// TIA Portal V19 export
FUNCTION_BLOCK "AreaGen_SafetyInterface_FB"   // FB6, LAD
// stored: Access Published, MemoryReserve 100, SetENOAutomatically false
   VAR_INPUT
      AreaInterface1 : "AreaInterface";
      AreaInterface2 : "AreaInterface";
      AreaInterface3 : "AreaInterface";
      AreaInterface4 : "AreaInterface";
   END_VAR
   VAR_OUTPUT
      MachineInterface1 : "MachineInterface";
      MachineInterface2 : "MachineInterface";
      MachineInterface3 : "MachineInterface";
      MachineInterface4 : "MachineInterface";
   END_VAR
   VAR
      Alarm : Struct
         G { ExternalAccessible := 'False'; ExternalVisible := 'False'; ExternalWritable := 'False'} : Struct
            EStop : Struct
               Area01 : Bool;
               Area02 : Bool;
               Area03 : Bool;
            END_STRUCT;
            FIO_Passivation : Struct
               Module_412A1 : Bool;
               Module_468A1 : Bool;
               Module_468A2 : Bool;
               Module_468A3 : Bool;
               Module_468A4 : Bool;
               Module_468A5 : Bool;
               Module_468A6 : Bool;
               Module_468A7 : Bool;
               Module_468A8 : Bool;
               Module_470A1 : Bool;
               Module_470A2 : Bool;
               Module_471A1 : Bool;
               Module_471A2 : Bool;
               Module_472A1 : Bool;
               Module_495A1 : Bool;
               Module_495A2 : Bool;
               Module_495A3 : Bool;
               Module_515A1 : Bool;
               Module_515A2 : Bool;
               Module_535A1 : Bool;
               Module_535A2 : Bool;
               Module_536A1 : Bool;
               Module_555A1 : Bool;
               Module_556A1 : Bool;
            END_STRUCT;
            FDBACK_Error : Struct
               F_Valve_Air_Gen_Contattore : Bool;
               F_Valve_Air_Gen_Cursore : Bool;
            END_STRUCT;
         END_STRUCT;
         Area01 { ExternalAccessible := 'False'; ExternalVisible := 'False'; ExternalWritable := 'False'} : Struct
            FDBACK_Error : Struct
               SafetyValve_CoilCar : Struct
                  FDO_FBK_ERROR : Bool;
                  EV_SAFETY_FBK_WARNING : Bool;
               END_STRUCT;
               SafetyValve_DecoilersHorizRotation : Struct
                  FDO_FBK_ERROR : Bool;
                  EV_SAFETY_FBK_WARNING : Bool;
               END_STRUCT;
               SafetyValve_Decoiler1 : Struct
                  FDO_FBK_ERROR : Bool;
                  EV_SAFETY_FBK_WARNING : Bool;
               END_STRUCT;
               SafetyValve_Decoiler2 : Struct
                  FDO_FBK_ERROR : Bool;
                  EV_SAFETY_FBK_WARNING : Bool;
               END_STRUCT;
               SafetyValve_Peeler : Struct
                  FDO_FBK_ERROR : Bool;
                  EV_SAFETY_FBK_WARNING : Bool;
               END_STRUCT;
               SafetyValve_JB_Cut_Rest : Struct
                  FDO_FBK_ERROR : Bool;
                  EV_SAFETY_FBK_WARNING : Bool;
               END_STRUCT;
               SafetyValve_JB_Cut_Work : Struct
                  FDO_FBK_ERROR : Bool;
                  EV_SAFETY_FBK_WARNING : Bool;
               END_STRUCT;
               HU_Decoilers_Motor_F_Contactor : Bool;
               HU_Area01_Motor_F_Contactor : Bool;
            END_STRUCT;
            S120_SafetyFaultActive : Struct
               CoilCar : Bool;
               DecoilersTranslation : Bool;
               Decoiler1 : Bool;
               Decoiler2 : Bool;
               Straightener : Bool;
               JBTorch : Bool;
               JBPinchRoll : Bool;
            END_STRUCT;
            UnathorizedOpen : Struct
               D01 : Bool;
               D02 : Bool;
               D03 : Bool;
               D04 : Bool;
               D05 : Bool;
               D07 : Bool;
            END_STRUCT;
         END_STRUCT;
         Area02 { ExternalAccessible := 'False'; ExternalVisible := 'False'; ExternalWritable := 'False'} : Struct
            FDBACK_Error : Struct
               F_Contactor_Rollformer_CambioFormato : Bool;
               F_Contactor_FinalCut_HU_Motor : Bool;
               F_Contactor_FinalCut_HU_Valve : Bool;
            END_STRUCT;
            S120_SafetyFaultActive : Struct
               Cassetta1_OP : Bool;
               Cassetta1_MOT : Bool;
               Cassetta2_OP : Bool;
               Cassetta2_MOT : Bool;
               Cassetta3_OP : Bool;
               Cassetta3_MOT : Bool;
               Rollformer : Bool;
               FAK_PusherAx : Bool;
               FlyCarriage : Bool;
               AccRolls1 : Bool;
               AccRolls2 : Bool;
               AccRolls3 : Bool;
            END_STRUCT;
            UnathorizedOpen : Struct
               D10 : Bool;
               D11 : Bool;
               D12 : Bool;
               D14 : Bool;
               D15 : Bool;
               D16 : Bool;
               D18 : Bool;
            END_STRUCT;
            PathTest_Rollformer : Bool;
         END_STRUCT;
         Area03_04 { ExternalAccessible := 'False'; ExternalVisible := 'False'; ExternalWritable := 'False'} : Struct
            FDBACK_Error : Struct
               F_Valve_Air_A0301_A0302_Contattore : Bool;
               F_Valve_Air_A0301_A0302_Cursore : Bool;
               F_Contactor_CambioFormato_Bordatrice : Bool;
               F_Contactor_Valvole_Pareggiatore_Testa : Bool;
               F_Contactor_Valvole_Pareggiatore_Coda : Bool;
               F_Valve_Air_A0302_A0303_Contattore : Bool;
               F_Valve_Air_A0302_A0303_Cursore : Bool;
               F_Valve_Air_A0304_Contattore : Bool;
               F_Valve_Air_A0304_Cursore : Bool;
            END_STRUCT;
            S120_SafetyFaultActive : Struct
               Trasporto : Bool;
               Ribaltatore : Bool;
               Spintore : Bool;
               Bordatrice : Bool;
               Rulliera_1 : Bool;
               Rulliera_2 : Bool;
               PareggiatoreCoda : Bool;
               PareggiatoreTesta : Bool;
               ManipolatoreCoda : Bool;
               ManipolatoreTesta : Bool;
               SpallaCoda : Bool;
               SpallaTesta : Bool;
               TraslazioneCoda : Bool;
               TraslazioneTesta : Bool;
               SollevamentoCoda : Bool;
               SollevamentoTesta : Bool;
               SostegnoAntiribCoda : Bool;
               SostegnoAntiribTesta : Bool;
               NavettaTesta : Bool;
               NavettaCoda : Bool;
            END_STRUCT;
            UnathorizedOpen : Struct
               D19 : Bool;
               D20 : Bool;
               D21 : Bool;
               D22 : Bool;
               D24 : Bool;
               D25 : Bool;
               D27 : Bool;
            END_STRUCT;
            PathTest_Bordatrice : Bool;
         END_STRUCT;
      END_STRUCT;
      Warning : Struct
         G { ExternalAccessible := 'False'; ExternalVisible := 'False'; ExternalWritable := 'False'} : Struct
            EStop_CC : Bool;
            EStop_A01_Front : Bool;
            EStop_A01_Rear : Bool;
            EStop_A02_Front : Bool;
            EStop_A02_Rear : Bool;
            EStop_A03_Front_1 : Bool;
            EStop_A03_Front_2 : Bool;
            EStop_A03_Front_3 : Bool;
            EStop_A03_Rear_1 : Bool;
            EStop_A03_Rear_2 : Bool;
            EStop_A03_Rear_3 : Bool;
         END_STRUCT;
         Area01 { ExternalAccessible := 'False'; ExternalVisible := 'False'; ExternalWritable := 'False'} : Struct
            Selectors : Struct
               Maintenance_MB1 : Bool;
            END_STRUCT;
            DoorOpened : Struct
               D01 : Bool;
               D02 : Bool;
               D03 : Bool;
               D04 : Bool;
               D05 : Bool;
               D06 : Bool;   // NOt EXIST
               D07 : Bool;
            END_STRUCT;
            DoorOpenRequest : Struct
               D01 : Bool;
               D02 : Bool;
               D03 : Bool;
               D04 : Bool;
               D05 : Bool;
               D06 : Bool;   // NOt EXIST
               D07 : Bool;
            END_STRUCT;
            DoorNotLocked : Struct
               D04 : Bool;
               D05 : Bool;
               D07 : Bool;
            END_STRUCT;
         END_STRUCT;
         Area02 { ExternalAccessible := 'False'; ExternalVisible := 'False'; ExternalWritable := 'False'} : Struct
            Selectors : Struct
               Maintenance_MB2 : Bool;
            END_STRUCT;
            Feedback : Struct
               F_Valve_Area02_HU : Bool;
            END_STRUCT;
            DoorOpened : Struct
               D10 : Bool;
               D11 : Bool;
               D12 : Bool;
               D14 : Bool;
               D15 : Bool;
               D16 : Bool;
               D18 : Bool;
            END_STRUCT;
            DoorOpenRequest : Struct
               D10 : Bool;
               D11 : Bool;
               D12 : Bool;
               D14 : Bool;
               D15 : Bool;
               D16 : Bool;
               D18 : Bool;
            END_STRUCT;
            PathTest_Rollformer : Bool;
         END_STRUCT;
         Area03_04 { ExternalAccessible := 'False'; ExternalVisible := 'False'; ExternalWritable := 'False'} : Struct
            Selectors : Struct
               Maintenance_MB3 : Bool;
            END_STRUCT;
            DoorOpened : Struct
               D18 : Bool;
               D19 : Bool;
               D20 : Bool;
               D21 : Bool;
               D22 : Bool;
               D24 : Bool;
               D25 : Bool;
               D27 : Bool;
            END_STRUCT;
            DoorOpenRequest : Struct
               D16 : Bool;
               D18 : Bool;
               D19 : Bool;
               D20 : Bool;
               D21 : Bool;
               D22 : Bool;
               D24 : Bool;
               D25 : Bool;
               D27 : Bool;
            END_STRUCT;
            DoorNotLocked : Struct
               D16 : Bool;
               D19 : Bool;
               D20 : Bool;
               D21 : Bool;
               D25 : Bool;
               D27 : Bool;
            END_STRUCT;
            PathTest_Bodatrice : Bool;
         END_STRUCT;
         NoAutReady : Bool;
      END_STRUCT;
      HMI : Struct
         PbResetEletricDoor : Bool;
         LpResetEletricDoor : Bool;
      END_STRUCT;
      TON_ResetEletricDoor : TON_TIME;
      AreaG_Safety { S7_SetPoint := 'True'} : "AreaG_SafetyInterface_FB";
      Area01_Safety { S7_SetPoint := 'True'} : "Area01_SafetyInterface_FB";
      Area02_Safety { S7_SetPoint := 'True'} : "Area02_SafetyInterface_FB";
      Area03_04_Safety { S7_SetPoint := 'True'} : "Area03_04_SafetyInterface_FB";
   END_VAR
   VAR_TEMP
      Rst : Bool;
      WarningPresebce : Bool;
   END_VAR
BEGIN

REGION Network 1: Reset alarms
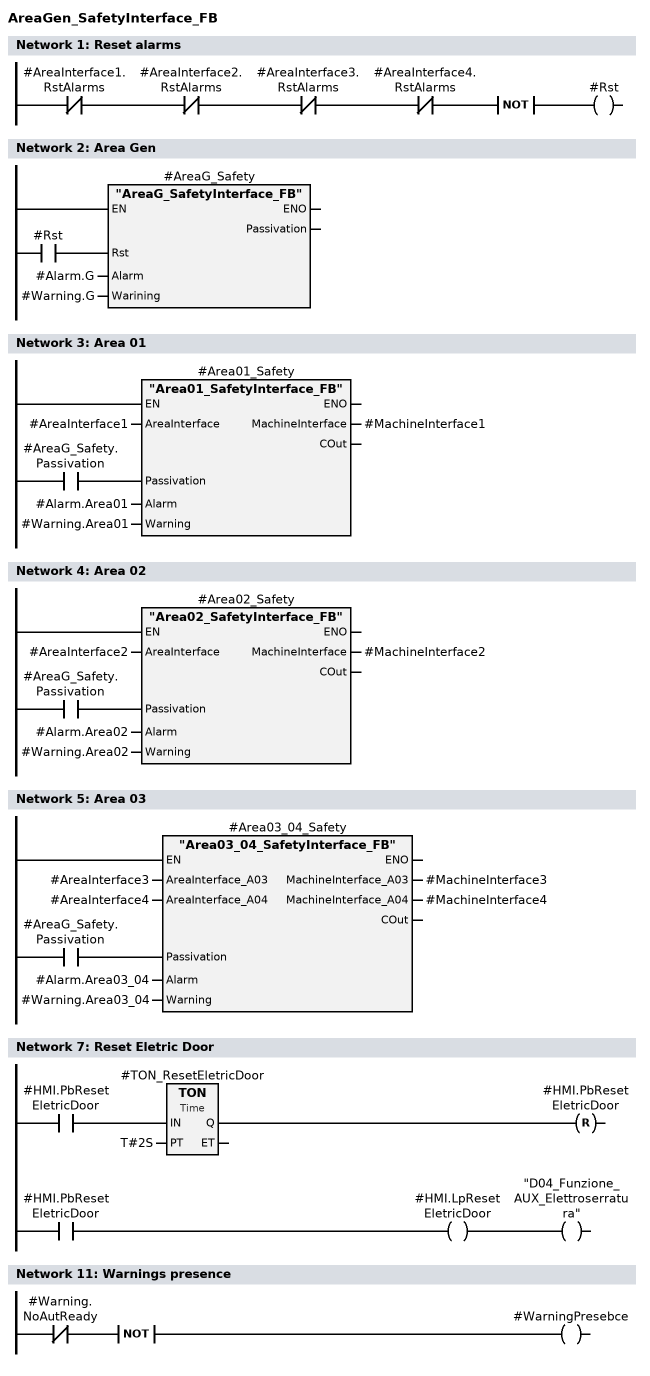
   RUNG wire#powerrail
      I_Contact( #AreaInterface1.RstAlarms )
      I_Contact( #AreaInterface2.RstAlarms )
      I_Contact( #AreaInterface3.RstAlarms )
      I_Contact( #AreaInterface4.RstAlarms )
      Not()
      Coil( #Rst )
   END_RUNG
   // the same network as SCL:
   #Rst := NOT (NOT #AreaInterface1.RstAlarms AND NOT #AreaInterface2.RstAlarms AND NOT #AreaInterface3.RstAlarms AND NOT #AreaInterface4.RstAlarms);
END_REGION

REGION Network 2: Area Gen
   RUNG wire#powerrail
      #AreaG_Safety(Rst := wire#w1, Alarm := #Alarm.G, Warining := #Warning.G, Passivation =>)
   END_RUNG
   RUNG wire#powerrail
      Contact( #Rst )
   END_RUNG wire#w1
   // the same network as SCL:
   #AreaG_Safety(Rst := #Rst, Alarm := #Alarm.G, Warining := #Warning.G);   // "AreaG_SafetyInterface_FB"
END_REGION

REGION Network 3: Area 01
   RUNG wire#powerrail
      #Area01_Safety(Passivation := wire#w1, AreaInterface := #AreaInterface1, Alarm := #Alarm.Area01, Warning := #Warning.Area01, MachineInterface => #MachineInterface1, COut =>)
   END_RUNG
   RUNG wire#powerrail
      Contact( #AreaG_Safety.Passivation )
   END_RUNG wire#w1
   // the same network as SCL:
   #Area01_Safety(AreaInterface := #AreaInterface1,   // "Area01_SafetyInterface_FB"
                  Passivation := #AreaG_Safety.Passivation,
                  Alarm := #Alarm.Area01,
                  Warning := #Warning.Area01,
                  MachineInterface => #MachineInterface1);
END_REGION

REGION Network 4: Area 02
   RUNG wire#powerrail
      #Area02_Safety(Passivation := wire#w1, AreaInterface := #AreaInterface2, Alarm := #Alarm.Area02, Warning := #Warning.Area02, MachineInterface => #MachineInterface2, COut =>)
   END_RUNG
   RUNG wire#powerrail
      Contact( #AreaG_Safety.Passivation )
   END_RUNG wire#w1
   // the same network as SCL:
   #Area02_Safety(AreaInterface := #AreaInterface2,   // "Area02_SafetyInterface_FB"
                  Passivation := #AreaG_Safety.Passivation,
                  Alarm := #Alarm.Area02,
                  Warning := #Warning.Area02,
                  MachineInterface => #MachineInterface2);
END_REGION

REGION Network 5: Area 03
   RUNG wire#powerrail
      #Area03_04_Safety(Passivation := wire#w1, AreaInterface_A03 := #AreaInterface3, AreaInterface_A04 := #AreaInterface4, Alarm := #Alarm.Area03_04, Warning := #Warning.Area03_04, MachineInterface_A03 => #MachineInterface3, MachineInterface_A04 => #MachineInterface4, COut =>)
   END_RUNG
   RUNG wire#powerrail
      Contact( #AreaG_Safety.Passivation )
   END_RUNG wire#w1
   // the same network as SCL:
   #Area03_04_Safety(AreaInterface_A03 := #AreaInterface3,   // "Area03_04_SafetyInterface_FB"
                     AreaInterface_A04 := #AreaInterface4,
                     Passivation := #AreaG_Safety.Passivation,
                     Alarm := #Alarm.Area03_04,
                     Warning := #Warning.Area03_04,
                     MachineInterface_A03 => #MachineInterface3,
                     MachineInterface_A04 => #MachineInterface4);
END_REGION

REGION Network 7: Reset Eletric Door
   RUNG wire#powerrail
      Contact( #HMI.PbResetEletricDoor )
      { S7_Templates := "time_type := Time" } #TON_ResetEletricDoor.TON(pt := T#2S, et =>)
      R_Coil( #HMI.PbResetEletricDoor )
   END_RUNG
   RUNG wire#powerrail
      Contact( #HMI.PbResetEletricDoor )
      Coil( #HMI.LpResetEletricDoor )
      Coil( "D04_Funzione_AUX_Elettroserratura" )
   END_RUNG
   // the same network as SCL:
   #TON_ResetEletricDoor(IN := #HMI.PbResetEletricDoor, PT := T#2S);   // TON
   IF #TON_ResetEletricDoor.Q THEN #HMI.PbResetEletricDoor := FALSE; END_IF;
   #HMI.LpResetEletricDoor := #HMI.PbResetEletricDoor;
   "D04_Funzione_AUX_Elettroserratura" := #HMI.PbResetEletricDoor;
END_REGION

REGION Network 9: <<< MACHINE STATUS >>>
END_REGION

REGION Network 10: Standstill
END_REGION

REGION Network 11: Warnings presence
   RUNG wire#powerrail
      I_Contact( #Warning.NoAutReady )
      Not()
      Coil( #WarningPresebce )
   END_RUNG
   // the same network as SCL:
   #WarningPresebce := NOT (NOT #Warning.NoAutReady);
END_REGION

REGION Network 12 (SCL): Collect machine to zone interface 2
   (*
   #MachineInterface2.AutReady := #AreaInterface2.Aut AND NOT #Sts.AlarmsPresence;
   #MachineInterface2.Aborting := #Sts.AlarmsPresence;
   #MachineInterface2.MotionsStandStill := #Sts.Standstill;
   #MachineInterface2.AckStopInPhase := #AreaInterface2.StopInPhase;
   #MachineInterface2.AckStopProgrammed := #AreaInterface2.StopProgrammed;
   #MachineInterface2.AlarmsPresence := #Sts.AlarmsPresence;
   #MachineInterface2.WarningPresence := #Sts.WarningsPresence;
   *)
END_REGION

REGION Network 13 (SCL): Collect machine to zone interface 3
   (*
   #MachineInterface3.AutReady := #AreaInterface3.Aut AND NOT #Sts.AlarmsPresence;
   #MachineInterface3.Aborting := #Sts.AlarmsPresence;
   #MachineInterface3.MotionsStandStill := #Sts.Standstill;
   #MachineInterface3.AckStopInPhase := #AreaInterface3.StopInPhase;
   #MachineInterface3.AckStopProgrammed := #AreaInterface3.StopProgrammed;
   #MachineInterface3.AlarmsPresence := #Sts.AlarmsPresence;
   #MachineInterface3.WarningPresence := #Sts.WarningsPresence;
   *)
END_REGION

REGION Network 14 (SCL): Warning Machine not ready for automatic
   IF (#AreaInterface1.CheckAutReady AND NOT #MachineInterface1.AutReady)
       OR
       (#AreaInterface2.CheckAutReady AND NOT #MachineInterface2.AutReady)
       OR
       (#AreaInterface3.CheckAutReady AND NOT #MachineInterface3.AutReady)
   THEN
       #Warning.NoAutReady := TRUE;
   ELSIF #Rst
   THEN
       #Warning.NoAutReady := FALSE;
   END_IF;
END_REGION
END_FUNCTION_BLOCK
